// TIA Portal V18 export
DATA_BLOCK "prePreviousValues"   // DB22
{ S7_Optimized_Access := 'TRUE' }
// stored: InstanceOfName UDT_actualValues, InstanceOfType UDT
"UDT_actualValues"
   // VAR RETAIN
   //    target { ExternalVisible := 'False'; ExternalWritable := 'False'} : DInt;
   //    actual { ExternalVisible := 'False'; ExternalWritable := 'False'} : DInt;
   //    ok { ExternalVisible := 'False'; ExternalWritable := 'False'} : DInt;
   //    difference { ExternalVisible := 'False'; ExternalWritable := 'False'} : DInt;
   //    counterTactTime { ExternalVisible := 'False'; ExternalWritable := 'False'} : DInt;
   //    state { ExternalVisible := 'False'; ExternalWritable := 'False'} : DInt;
   //    taktTime : DInt;
   // END_VAR
BEGIN
END_DATA_BLOCK
